// TIA Portal V21 export
VAR_GLOBAL   // PLC tag table "PastorizzatoreReciveDigitali"
END_VAR
VAR_GLOBAL CONSTANT   // user constants
   K_SegnaleDaPastorizzatore_Marcia : Int := 1;
END_VAR
